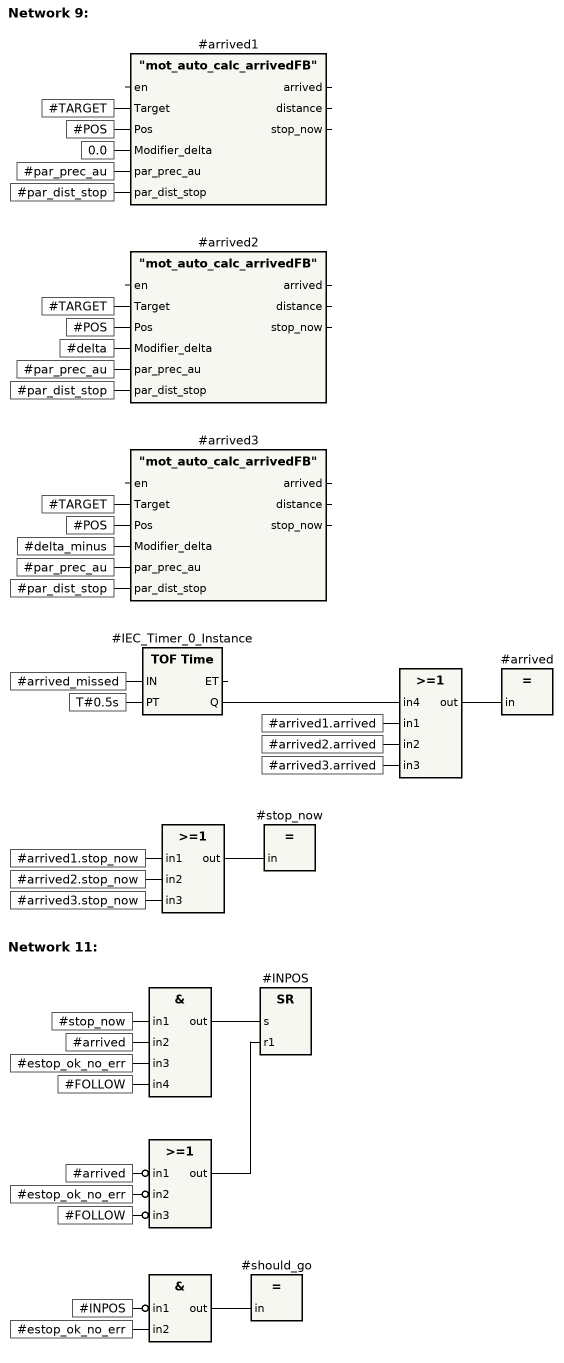
   #arrived1(Target := #TARGET,   // "mot_auto_calc_arrivedFB"
             Pos := #POS,
             Modifier_delta := 0.0,
             par_prec_au := #par_prec_au,
             par_dist_stop := #par_dist_stop);
   #arrived2(Target := #TARGET,   // "mot_auto_calc_arrivedFB"
             Pos := #POS,
             Modifier_delta := #delta,
             par_prec_au := #par_prec_au,
             par_dist_stop := #par_dist_stop);
   #arrived3(Target := #TARGET,   // "mot_auto_calc_arrivedFB"
             Pos := #POS,
             Modifier_delta := #delta_minus,
             par_prec_au := #par_prec_au,
             par_dist_stop := #par_dist_stop);
   #IEC_Timer_0_Instance(IN := #arrived_missed, PT := T#0.5s);   // TOF
   #arrived := #IEC_Timer_0_Instance.Q OR #arrived1.arrived OR #arrived2.arrived OR #arrived3.arrived;
   #stop_now := #arrived1.stop_now OR #arrived2.stop_now OR #arrived3.stop_now;
END_REGION

REGION Network 11
   IF #stop_now AND #arrived AND #estop_ok_no_err AND #FOLLOW THEN
       #INPOS := TRUE;   // SR flip-flop
   END_IF;
   IF NOT #arrived OR NOT #estop_ok_no_err OR NOT #FOLLOW THEN #INPOS := FALSE; END_IF;
   #should_go := NOT #INPOS AND #estop_ok_no_err;
END_REGION

REGION Network 12
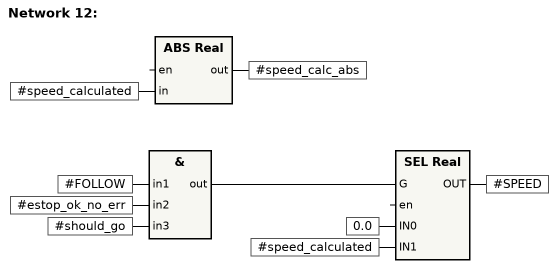
   #speed_calc_abs := ABS(#speed_calculated);
   #SPEED := SEL(G := #FOLLOW AND #estop_ok_no_err AND #should_go, IN0 := 0.0, IN1 := #speed_calculated);
END_REGION
END_FUNCTION_BLOCK

FUNCTION_BLOCK "mot_auto_calc_arrivedFB"   // FB57, FBD
{ S7_Optimized_Access := 'TRUE' }
VERSION : 0.1
// stored: AutoNumber true, IsIECCheckEnabled false, IsRetainMemResEnabled false, MemoryReserve 100, SetENOAutomatically false, UDAEnableTagReadback false
   VAR_INPUT
      Target { ExternalAccessible := 'False'; ExternalVisible := 'False'; ExternalWritable := 'False'} : Real;
      Pos { ExternalAccessible := 'False'; ExternalVisible := 'False'; ExternalWritable := 'False'} : Real;
      Modifier_delta { ExternalAccessible := 'False'; ExternalVisible := 'False'; ExternalWritable := 'False'} : Real;
      par_prec_au { ExternalAccessible := 'False'; ExternalVisible := 'False'; ExternalWritable := 'False'} : Real;
      par_dist_stop { ExternalAccessible := 'False'; ExternalVisible := 'False'; ExternalWritable := 'False'} : Real;
   END_VAR
   VAR_OUTPUT
      arrived { ExternalAccessible := 'False'; ExternalVisible := 'False'; ExternalWritable := 'False'} : Bool;
      distance { ExternalAccessible := 'False'; ExternalVisible := 'False'; ExternalWritable := 'False'} : Real;
      stop_now { ExternalAccessible := 'False'; ExternalVisible := 'False'; ExternalWritable := 'False'} : Bool;
   END_VAR
BEGIN

REGION Network 2 (SCL)
   #distance := #Target - (#Pos + #Modifier_delta);

   #arrived := ABS(#distance) <= #par_prec_au;

   #stop_now := ABS(#distance) <= #par_dist_stop;
END_REGION
END_FUNCTION_BLOCK

FUNCTION_BLOCK "mot_speed_abs_slowly_accelerated"   // FB67, FBD
{ S7_Optimized_Access := 'TRUE' }
VERSION : 0.1
// stored: AutoNumber true, IsIECCheckEnabled false, IsRetainMemResEnabled false, MemoryReserve 100, SetENOAutomatically false, UDAEnableTagReadback false
   VAR_INPUT
      ALLOWED : Bool;
      set_speed_abs : Real;
      v_absMax : Real;
      t_acc : Real;
   END_VAR
   VAR_OUTPUT
      speed_accelerated_slowly_abs : Real;
   END_VAR
   VAR_TEMP
      cycle_time_s : Real;
      acceleration : Real;
      accleration_per_cycle : Real;
   END_VAR
BEGIN

REGION Network 2 (SCL)
   #cycle_time_s := "_MAIN_DB".CLOCK_S_P_SCAN;
   IF #t_acc > 0 THEN
       #acceleration := #v_absMax / #t_acc;
       #accleration_per_cycle := #acceleration * #cycle_time_s;
       IF NOT #ALLOWED OR #set_speed_abs = 0 THEN
           #speed_accelerated_slowly_abs := #set_speed_abs;
       ELSE
           #speed_accelerated_slowly_abs := LIMIT(MN := 0, IN := #speed_accelerated_slowly_abs + #accleration_per_cycle, MX := #set_speed_abs);
       END_IF;
   ELSE
       #speed_accelerated_slowly_abs := #set_speed_abs;
   END_IF;
END_REGION
END_FUNCTION_BLOCK

FUNCTION_BLOCK "mot_speed_wdir_slowly_accelerated"   // FB68, FBD
{ S7_Optimized_Access := 'TRUE' }
VERSION : 0.1
// stored: AutoNumber true, IsIECCheckEnabled false, IsRetainMemResEnabled false, MemoryReserve 100, SetENOAutomatically false, UDAEnableTagReadback false
   VAR_INPUT
      ALLOWED : Bool;
      set_speed__wdir : Real;
      v_absMax : Real;
      t_acc : Real;
      STOP_NOW : Bool;
   END_VAR
   VAR_OUTPUT
      speed_accelerated_slowly_wdir : Real;
   END_VAR
   VAR
      speed_is_zero : Bool;
      speed_is_zero_was : Bool;
      speed_is_zero_CLK : Bool;
   END_VAR
   VAR_TEMP
      cycle_time_s : Real;
      acceleration : Real;
      accleration_per_cycle : Real;
   END_VAR
BEGIN

REGION Network 2 (SCL)
   #speed_is_zero := #set_speed__wdir = 0;
   #speed_is_zero_CLK := false;//AND #speed_is_zero AND NOT #speed_is_zero_was; 
   #speed_is_zero_was := #speed_is_zero ;
END_REGION

REGION Network 3 (SCL)
   #cycle_time_s := "_MAIN_DB".CLOCK_S_P_SCAN;
   IF #t_acc > 0 AND NOT #STOP_NOW THEN
       #acceleration := #v_absMax / #t_acc;
       #accleration_per_cycle := #acceleration * #cycle_time_s;
       IF NOT #ALLOWED OR #speed_is_zero_CLK  THEN
           #speed_accelerated_slowly_wdir := #set_speed__wdir;
       ELSE
           IF #speed_accelerated_slowly_wdir < #set_speed__wdir THEN
               #speed_accelerated_slowly_wdir := MIN(IN1 := #speed_accelerated_slowly_wdir + #accleration_per_cycle, IN2 := #set_speed__wdir);
           ELSE 
               #speed_accelerated_slowly_wdir := MAX(IN1 := #speed_accelerated_slowly_wdir - #accleration_per_cycle,IN2 := #set_speed__wdir);
           END_IF;
       END_IF;
   ELSE
       #speed_accelerated_slowly_wdir := #set_speed__wdir;
   END_IF;
END_REGION
END_FUNCTION_BLOCK

FUNCTION_BLOCK "manual_analog"   // FB7, FBD
{ S7_Optimized_Access := 'TRUE' }
VERSION : 0.1
// stored: AutoNumber true, IsIECCheckEnabled false, IsRetainMemResEnabled false, MemoryReserve 100, SetENOAutomatically false, UDAEnableTagReadback false
   VAR_INPUT
      ALLOWED : Bool;
      ALLOWED_ONLY_IN_OVERRIDE : Bool;
      OVERRIDE_NOW : Bool;
      isMultiturn : Bool;
      POS : Real;
      SET_SPEED : Real;
      xFwdOk : Bool;
      xRevOk : Bool;
      clibrated : Bool;
      par_spd_absmax : Real := 1000.0;
      par_dist_absmax : Real := 100.0;
      par_speed_crawl : Real;
      par_dist_crawl : Real;
      par_dist_stop : Real := 10.0;
      par_spd_blind : Real := 500.0;
      par_fwd_limit : Real := 10000.0;
      par_rev_limit : Real := 0.0;
      par_t_acc : Real;
   END_VAR
   VAR_OUTPUT
      SPEED : Real;
      ER_settings : Bool;
      er_ws : WString;
   END_VAR
   VAR
      speed_slowly_accelerated : Real;
      mot_speed_wdir_slowly_accelerated_Instance { S7_SetPoint := 'True'} : "mot_speed_wdir_slowly_accelerated";
   END_VAR
   VAR_TEMP
      speed_calculated : Real;
      speed_calc_abs : Real;
      estop_ok_no_err : Bool;
      blind : Bool;
      set_spd_loc : Real;
   END_VAR
   VAR CONSTANT
      erwsnoer : WString := WSTRING#'no er';
      erws1 : WString := WSTRING#'lim fwd = rev';
      erws2 : WString := WSTRING#'#par_dist_fast 0';
      erws3 : WString := WSTRING#'#par_spd_absmax';
   END_VAR
   VAR_TEMP   // added for the SCL form of the ladder/FBD networks
      _w1 : Bool;
      _w2 : Bool;
   END_VAR
BEGIN

REGION Network 1
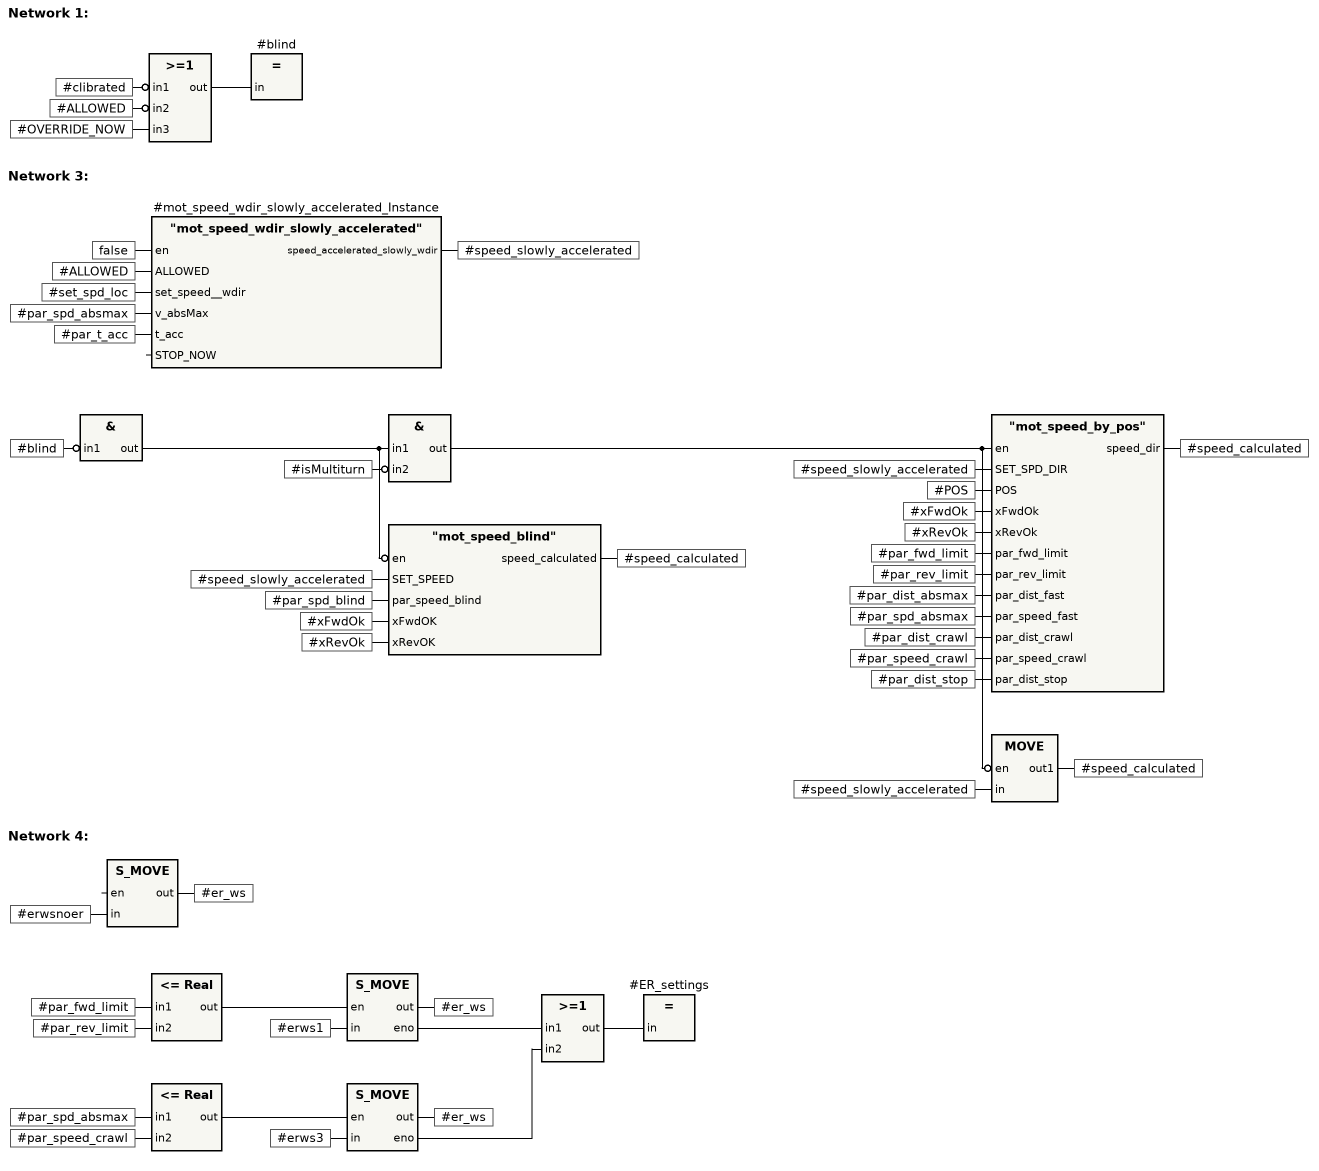
   #blind := NOT #clibrated OR NOT #ALLOWED OR #OVERRIDE_NOW;
END_REGION

REGION Network 2 (SCL)
   #speed_slowly_accelerated := #set_spd_loc := LIMIT(IN:=#SET_SPEED,MN:=-#par_spd_absmax,MX:=#par_spd_absmax);
   //#SET_SPEED*#par_spd_fast
END_REGION

REGION Network 3
   IF false THEN
       #mot_speed_wdir_slowly_accelerated_Instance(ALLOWED := #ALLOWED,   // "mot_speed_wdir_slowly_accelerated"
                               set_speed__wdir := #set_spd_loc,
                               v_absMax := #par_spd_absmax,
                               t_acc := #par_t_acc,
                               speed_accelerated_slowly_wdir => #speed_slowly_accelerated);
   END_IF;
   #_w1 := NOT #blind AND NOT #isMultiturn;
   IF #_w1 THEN
       "mot_speed_by_pos"(SET_SPD_DIR := #speed_slowly_accelerated,
                          POS := #POS,
                          xFwdOk := #xFwdOk,
                          xRevOk := #xRevOk,
                          par_fwd_limit := #par_fwd_limit,
                          par_rev_limit := #par_rev_limit,
                          par_dist_fast := #par_dist_absmax,
                          par_speed_fast := #par_spd_absmax,
                          par_dist_crawl := #par_dist_crawl,
                          par_speed_crawl := #par_speed_crawl,
                          par_dist_stop := #par_dist_stop,
                          speed_dir => #speed_calculated);
   END_IF;
   IF NOT #_w1 THEN #speed_calculated := #speed_slowly_accelerated; END_IF;
   IF NOT (NOT #blind) THEN
       "mot_speed_blind"(SET_SPEED := #speed_slowly_accelerated,
                         par_speed_blind := #par_spd_blind,
                         xFwdOK := #xFwdOk,
                         xRevOK := #xRevOk,
                         speed_calculated => #speed_calculated);
   END_IF;
END_REGION

REGION Network 4
   #er_ws := #erwsnoer;
   #_w1 := #par_fwd_limit <= #par_rev_limit;
   IF #_w1 THEN #er_ws := #erws1; END_IF;
   #_w2 := #par_spd_absmax <= #par_speed_crawl;
   IF #_w2 THEN #er_ws := #erws3; END_IF;
   #ER_settings := #_w1 OR #_w2;
END_REGION

REGION Network 5
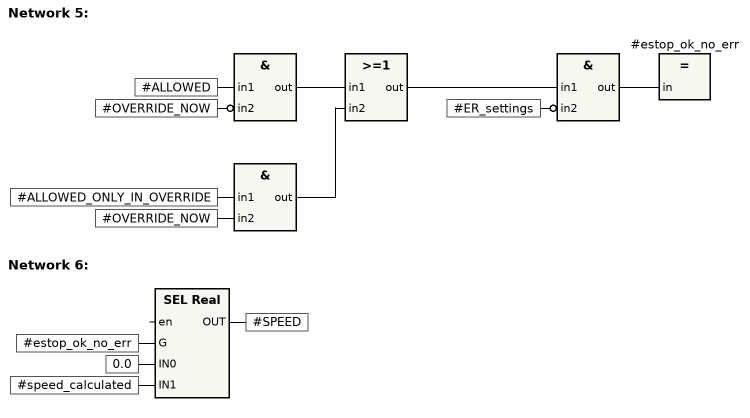
   #estop_ok_no_err := ((#ALLOWED AND NOT #OVERRIDE_NOW) OR (#ALLOWED_ONLY_IN_OVERRIDE AND #OVERRIDE_NOW)) AND NOT #ER_settings;
END_REGION

REGION Network 6
   #SPEED := SEL(G := #estop_ok_no_err, IN0 := 0.0, IN1 := #speed_calculated);
END_REGION
END_FUNCTION_BLOCK

FUNCTION "mot_speed_blind" : Void   // FC11, FBD
{ S7_Optimized_Access := 'TRUE' }
VERSION : 0.1
// stored: AutoNumber true, IsIECCheckEnabled false, SetENOAutomatically false, UDAEnableTagReadback false
   VAR_INPUT
      SET_SPEED : Real;
      par_speed_blind : Real;
      xFwdOK : Bool;
      xRevOK : Bool;
   END_VAR
   VAR_OUTPUT
      speed_calculated : Real;
   END_VAR
   VAR_TEMP
      go_fwd : Bool;
      go_rev : Bool;
   END_VAR
BEGIN

REGION Network 1
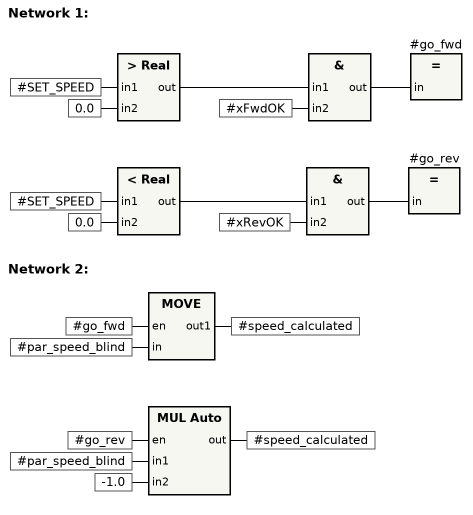
   #go_fwd := (#SET_SPEED > 0.0) AND #xFwdOK;
   #go_rev := (#SET_SPEED < 0.0) AND #xRevOK;
END_REGION

REGION Network 2
   IF #go_fwd THEN #speed_calculated := #par_speed_blind; END_IF;
   IF #go_rev THEN #speed_calculated := #par_speed_blind * (-1.0); END_IF;
END_REGION
END_FUNCTION

FUNCTION_BLOCK "enc_no_change_in_time"   // FB6, FBD
{ S7_Optimized_Access := 'TRUE' }
VERSION : 0.1
// stored: AutoNumber true, IsIECCheckEnabled false, IsRetainMemResEnabled false, MemoryReserve 100, SetENOAutomatically false, UDAEnableTagReadback false
   VAR_INPUT
      pt : Time := T#1s;
      FWD : Bool;
      REV : Bool;
      POS : Real;
   END_VAR
   VAR_OUTPUT
      ER_FWD : Bool;
      ER_REV : Bool;
   END_VAR
   VAR
      going_fwd { ExternalAccessible := 'False'; ExternalVisible := 'False'; ExternalWritable := 'False'} : Bool;
      going_rev { ExternalAccessible := 'False'; ExternalVisible := 'False'; ExternalWritable := 'False'} : Bool;
      going_not { ExternalAccessible := 'False'; ExternalVisible := 'False'; ExternalWritable := 'False'} : Bool;
      mem : Real;
      t_fwd { S7_SetPoint := 'True'} : TON_TIME;
      t_rev { S7_SetPoint := 'True'} : TON_TIME;
   END_VAR
BEGIN

REGION Network 1
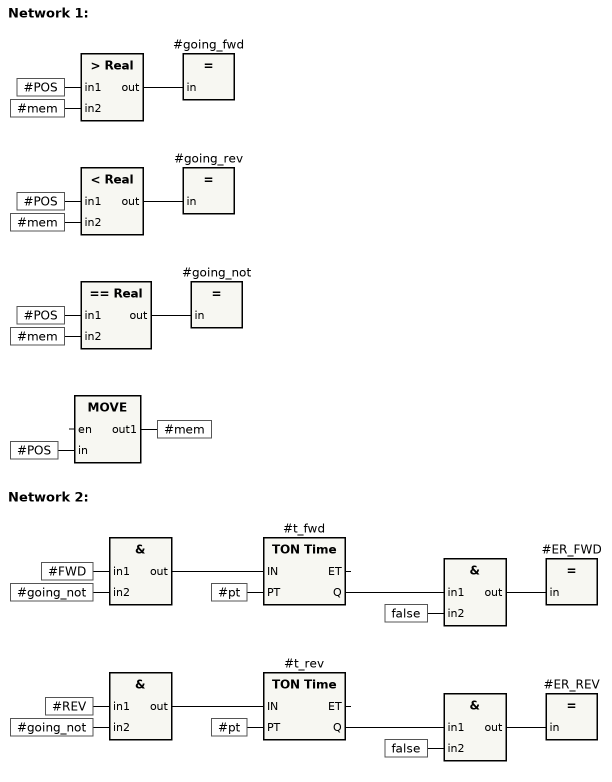
   #going_fwd := #POS > #mem;
   #going_rev := #POS < #mem;
   #going_not := #POS = #mem;
   #mem := #POS;
END_REGION

REGION Network 2
   #t_fwd(IN := #FWD AND #going_not, PT := #pt);   // TON
   #ER_FWD := #t_fwd.Q AND false;
   #t_rev(IN := #REV AND #going_not, PT := #pt);   // TON
   #ER_REV := #t_rev.Q AND false;
END_REGION
END_FUNCTION_BLOCK

FUNCTION_BLOCK "BRK_FB"   // FB21, FBD
{ S7_Optimized_Access := 'TRUE' }
VERSION : 0.1
// stored: AutoNumber true, IsIECCheckEnabled false, IsRetainMemResEnabled false, MemoryReserve 100, SetENOAutomatically false, UDAEnableTagReadback false
   VAR_INPUT
      SpeedZero : Bool;
      fwd : Bool;
      rev : Bool;
      pt : Time := T#100ms;
      error : Bool;
   END_VAR
   VAR_OUTPUT
      BRK_REL { ExternalAccessible := 'False'; ExternalVisible := 'False'; ExternalWritable := 'False'} : Bool;
   END_VAR
   VAR
      IEC_Timer_0_Instance { S7_SetPoint := 'True'} : TOF_TIME;
   END_VAR
BEGIN

REGION Network 2
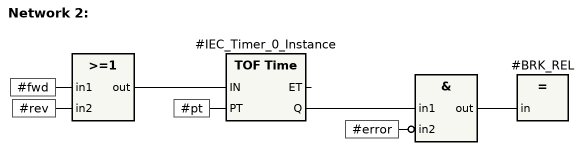
   #IEC_Timer_0_Instance(IN := #fwd OR #rev, PT := #pt);   // TOF
   #BRK_REL := #IEC_Timer_0_Instance.Q AND NOT #error;
END_REGION
END_FUNCTION_BLOCK

FUNCTION "f_ao_10V" : Int
{ S7_Optimized_Access := 'TRUE' }
VERSION : 0.1
   VAR_INPUT 
      "in 0.0-10.0" : Real;
   END_VAR

   VAR_TEMP 
      value_for_10V : Real;
      "r10.0" : Real;
   END_VAR


BEGIN
	#value_for_10V := 27648.0;(* tested FPY value 27175.0 *)
	#"r10.0" := 10.0;
	#f_ao_10V := DINT_TO_INT(
	                                 REAL_TO_DINT(
	                                              LIMIT(IN := #"in 0.0-10.0", MN := 0, MX := #"r10.0")
	                                              / #"r10.0" * #value_for_10V)
	);
END_FUNCTION

ORGANIZATION_BLOCK "Cyclic interrupt_axis_30ms"   // OB31, LAD, CyclicInterrupt
{ S7_Optimized_Access := 'TRUE' }
VERSION : 0.1
// stored: AutoNumber true, IsIECCheckEnabled false, SetENOAutomatically false
   VAR_INPUT
      Initial_Call : Bool;
      Event_Count : Int;
   END_VAR
BEGIN

REGION Network 1
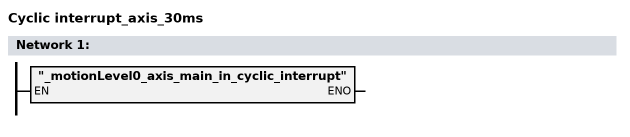
   RUNG wire#powerrail
      "_motionLevel0_axis_main_in_cyclic_interrupt"()
   END_RUNG
   // the same network as SCL:
   "_motionLevel0_axis_main_in_cyclic_interrupt"();
END_REGION
END_ORGANIZATION_BLOCK

FUNCTION "_motionLevel0_axis_main_in_cyclic_interrupt" : Void   // FC13, FBD
{ S7_Optimized_Access := 'TRUE' }
VERSION : 0.1
// stored: AutoNumber true, IsIECCheckEnabled false, SetENOAutomatically false, UDAEnableTagReadback false
   VAR_TEMP
      doors : Bool;
      "xray uses doors fwd closed mech" : Bool;
      "добавить блокировку вперед по световой завесе" : Bool;
      loc_dor_c_opn : Bool;
      loc_dor_c_cls : Bool;
      doorsWnOpnNAld : Bool;
      doorsWnClsNAld : Bool;
      ошибка_задания_искуственных_границ : Bool;
      динамическая_граница_y_rev : Real;
      динамическая_граница_y_fwd : Real;
      динамическая_граница_x_rev : Real;
      динамическая_граница_x_fwd : Real;
      манипулятор_не_мешает_дверям : Bool;
      doors_wnmanipulator : Bool;
   END_VAR
BEGIN

REGION Network 2
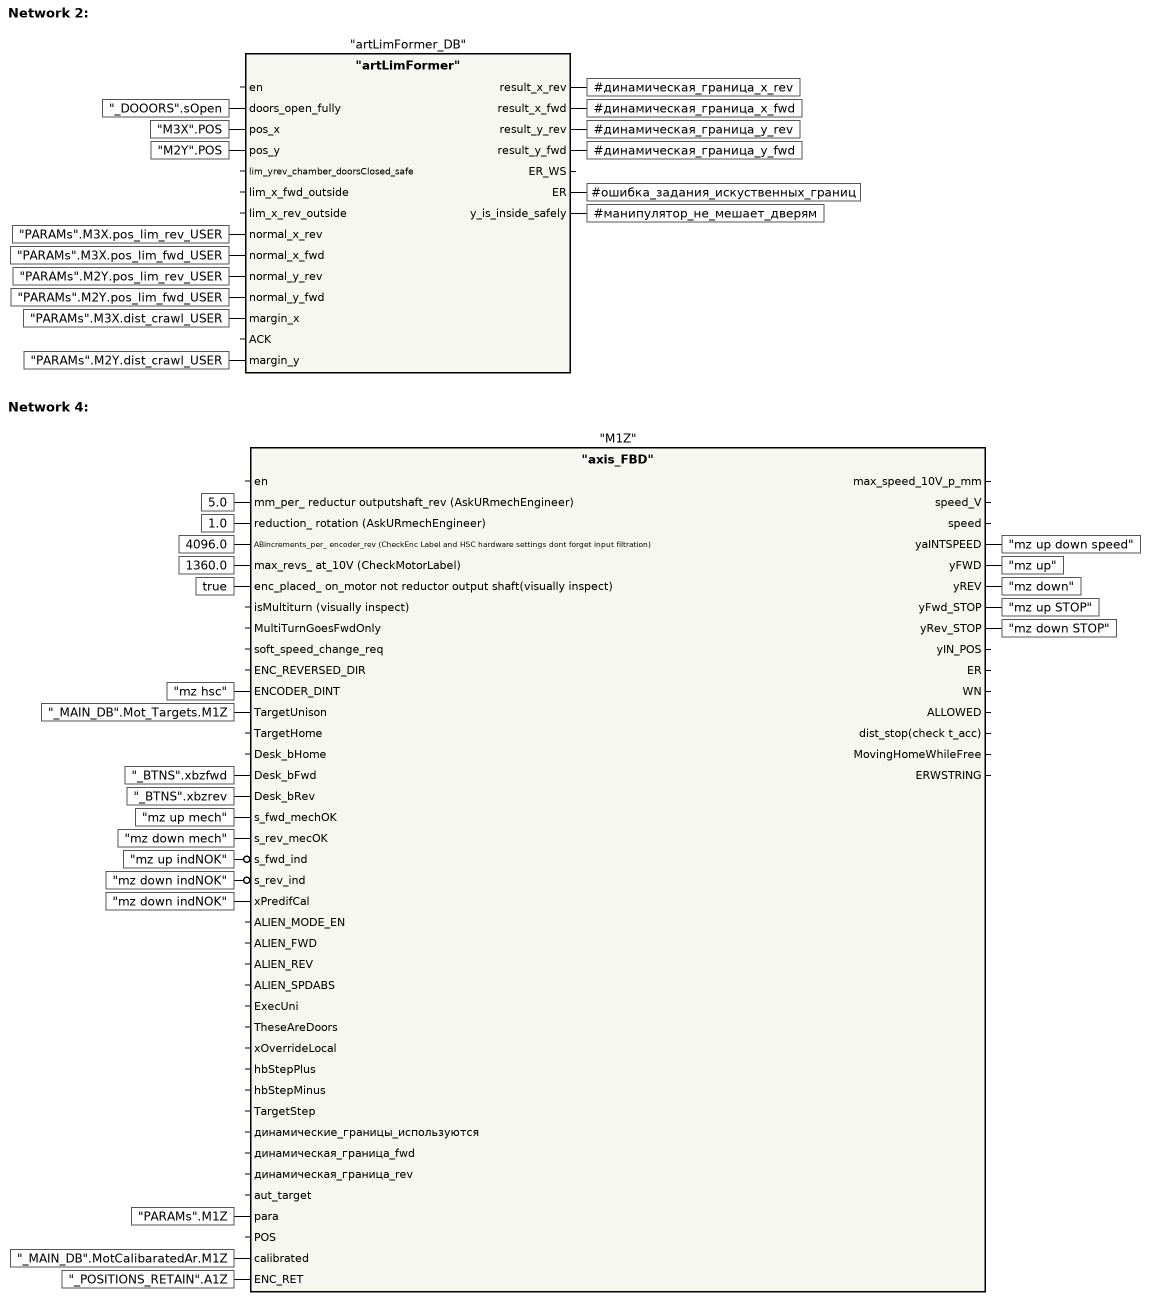
   "artLimFormer_DB"(doors_open_fully := "_DOOORS".sOpen,   // "artLimFormer"
                     pos_x := "M3X".POS,
                     pos_y := "M2Y".POS,
                     normal_x_rev := "PARAMs".M3X.pos_lim_rev_USER,
                     normal_x_fwd := "PARAMs".M3X.pos_lim_fwd_USER,
                     normal_y_rev := "PARAMs".M2Y.pos_lim_rev_USER,
                     normal_y_fwd := "PARAMs".M2Y.pos_lim_fwd_USER,
                     margin_x := "PARAMs".M3X.dist_crawl_USER,
                     margin_y := "PARAMs".M2Y.dist_crawl_USER,
                     result_x_rev => #динамическая_граница_x_rev,
                     result_x_fwd => #динамическая_граница_x_fwd,
                     result_y_rev => #динамическая_граница_y_rev,
                     result_y_fwd => #динамическая_граница_y_fwd,
                     ER => #ошибка_задания_искуственных_границ,
                     y_is_inside_safely => #манипулятор_не_мешает_дверям);
END_REGION

REGION Network 4
   "M1Z"("mm_per_ reductur outputshaft_rev (AskURmechEngineer)" := 5.0,   // "axis_FBD"
         "reduction_ rotation (AskURmechEngineer)" := 1.0,
         "ABincrements_per_ encoder_rev (CheckEnc Label and HSC hardware settings dont forget input filtration)" := 4096.0,
         "max_revs_ at_10V (CheckMotorLabel)" := 1360.0,
         "enc_placed_ on_motor not reductor output shaft(visually inspect)" := true,
         ENCODER_DINT := "mz hsc",
         TargetUnison := "_MAIN_DB".Mot_Targets.M1Z,
         Desk_bFwd := "_BTNS".xbzfwd,
         Desk_bRev := "_BTNS".xbzrev,
         s_fwd_mechOK := "mz up mech",
         s_rev_mecOK := "mz down mech",
         s_fwd_ind := NOT "mz up indNOK",
         s_rev_ind := NOT "mz down indNOK",
         xPredifCal := "mz down indNOK",
         para := "PARAMs".M1Z,
         calibrated := "_MAIN_DB".MotCalibaratedAr.M1Z,
         ENC_RET := "_POSITIONS_RETAIN".A1Z,
         yaINTSPEED => "mz up down speed",
         yFWD => "mz up",
         yREV => "mz down",
         yFwd_STOP => "mz up STOP",
         yRev_STOP => "mz down STOP");
END_REGION

REGION Network 5
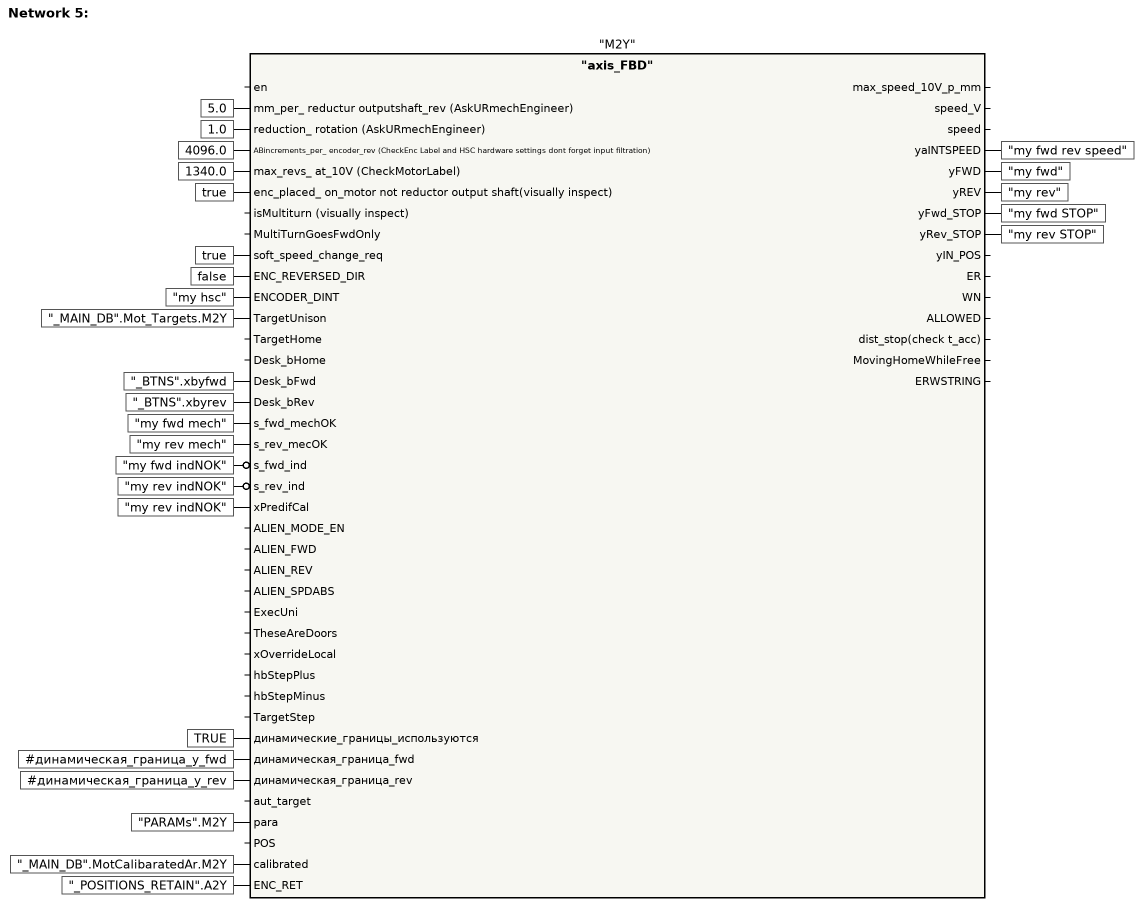
   "M2Y"("mm_per_ reductur outputshaft_rev (AskURmechEngineer)" := 5.0,   // "axis_FBD"
         "reduction_ rotation (AskURmechEngineer)" := 1.0,
         "ABincrements_per_ encoder_rev (CheckEnc Label and HSC hardware settings dont forget input filtration)" := 4096.0,
         "max_revs_ at_10V (CheckMotorLabel)" := 1340.0,
         "enc_placed_ on_motor not reductor output shaft(visually inspect)" := true,
         soft_speed_change_req := true,
         ENC_REVERSED_DIR := false,
         ENCODER_DINT := "my hsc",
         TargetUnison := "_MAIN_DB".Mot_Targets.M2Y,
         Desk_bFwd := "_BTNS".xbyfwd,
         Desk_bRev := "_BTNS".xbyrev,
         s_fwd_mechOK := "my fwd mech",
         s_rev_mecOK := "my rev mech",
         s_fwd_ind := NOT "my fwd indNOK",
         s_rev_ind := NOT "my rev indNOK",
         xPredifCal := "my rev indNOK",
         динамические_границы_используются := TRUE,
         динамическая_граница_fwd := #динамическая_граница_y_fwd,
         динамическая_граница_rev := #динамическая_граница_y_rev,
         para := "PARAMs".M2Y,
         calibrated := "_MAIN_DB".MotCalibaratedAr.M2Y,
         ENC_RET := "_POSITIONS_RETAIN".A2Y,
         yaINTSPEED => "my fwd rev speed",
         yFWD => "my fwd",
         yREV => "my rev",
         yFwd_STOP => "my fwd STOP",
         yRev_STOP => "my rev STOP");
END_REGION

REGION Network 6
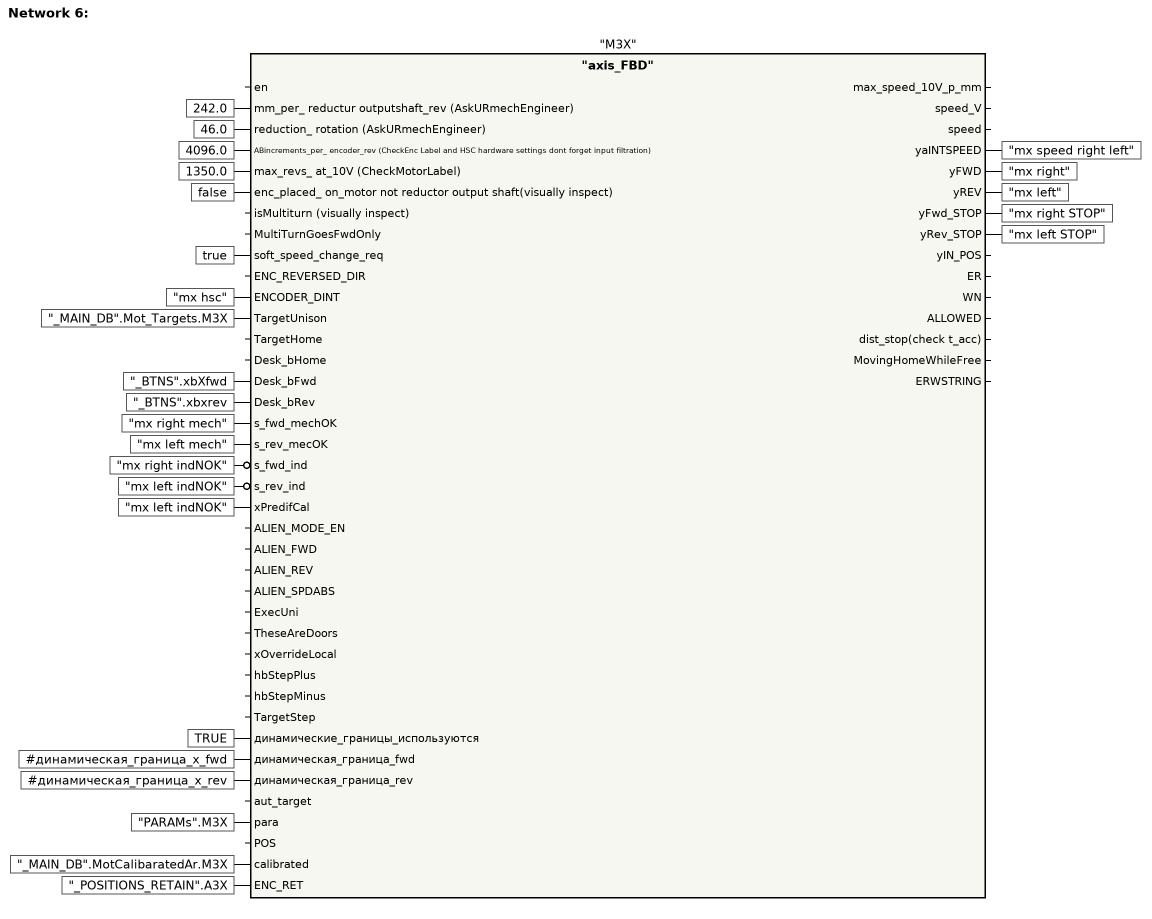
   "M3X"("mm_per_ reductur outputshaft_rev (AskURmechEngineer)" := 242.0,   // "axis_FBD"
         "reduction_ rotation (AskURmechEngineer)" := 46.0,
         "ABincrements_per_ encoder_rev (CheckEnc Label and HSC hardware settings dont forget input filtration)" := 4096.0,
         "max_revs_ at_10V (CheckMotorLabel)" := 1350.0,
         "enc_placed_ on_motor not reductor output shaft(visually inspect)" := false,
         soft_speed_change_req := true,
         ENCODER_DINT := "mx hsc",
         TargetUnison := "_MAIN_DB".Mot_Targets.M3X,
         Desk_bFwd := "_BTNS".xbXfwd,
         Desk_bRev := "_BTNS".xbxrev,
         s_fwd_mechOK := "mx right mech",
         s_rev_mecOK := "mx left mech",
         s_fwd_ind := NOT "mx right indNOK",
         s_rev_ind := NOT "mx left indNOK",
         xPredifCal := "mx left indNOK",
         динамические_границы_используются := TRUE,
         динамическая_граница_fwd := #динамическая_граница_x_fwd,
         динамическая_граница_rev := #динамическая_граница_x_rev,
         para := "PARAMs".M3X,
         calibrated := "_MAIN_DB".MotCalibaratedAr.M3X,
         ENC_RET := "_POSITIONS_RETAIN".A3X,
         yaINTSPEED => "mx speed right left",
         yFWD => "mx right",
         yREV => "mx left",
         yFwd_STOP => "mx right STOP",
         yRev_STOP => "mx left STOP");
END_REGION

REGION Network 7
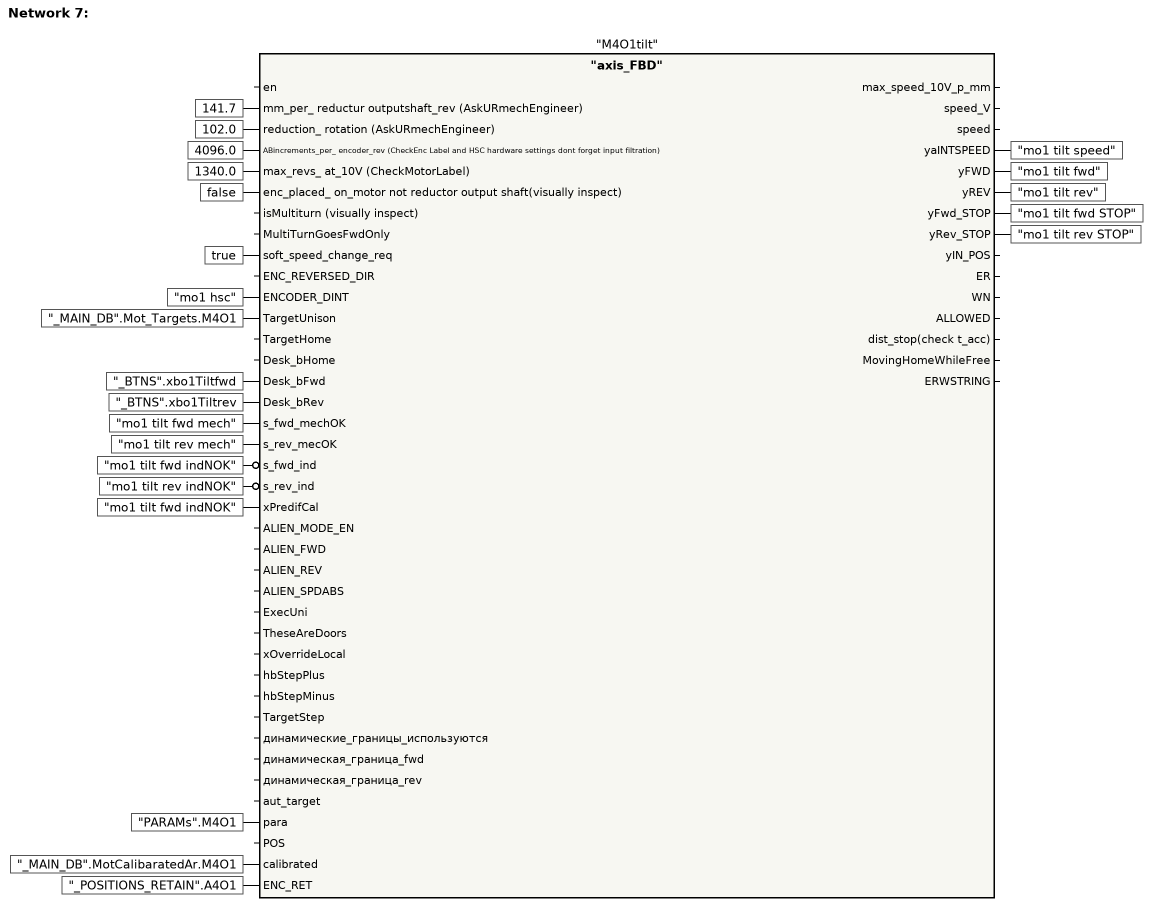
   "M4O1tilt"("mm_per_ reductur outputshaft_rev (AskURmechEngineer)" := 141.7,   // "axis_FBD"
              "reduction_ rotation (AskURmechEngineer)" := 102.0,
              "ABincrements_per_ encoder_rev (CheckEnc Label and HSC hardware settings dont forget input filtration)" := 4096.0,
              "max_revs_ at_10V (CheckMotorLabel)" := 1340.0,
              "enc_placed_ on_motor not reductor output shaft(visually inspect)" := false,
              soft_speed_change_req := true,
              ENCODER_DINT := "mo1 hsc",
              TargetUnison := "_MAIN_DB".Mot_Targets.M4O1,
              Desk_bFwd := "_BTNS".xbo1Tiltfwd,
              Desk_bRev := "_BTNS".xbo1Tiltrev,
              s_fwd_mechOK := "mo1 tilt fwd mech",
              s_rev_mecOK := "mo1 tilt rev mech",
              s_fwd_ind := NOT "mo1 tilt fwd indNOK",
              s_rev_ind := NOT "mo1 tilt rev indNOK",
              xPredifCal := "mo1 tilt fwd indNOK",
              para := "PARAMs".M4O1,
              calibrated := "_MAIN_DB".MotCalibaratedAr.M4O1,
              ENC_RET := "_POSITIONS_RETAIN".A4O1,
              yaINTSPEED => "mo1 tilt speed",
              yFWD => "mo1 tilt fwd",
              yREV => "mo1 tilt rev",
              yFwd_STOP => "mo1 tilt fwd STOP",
              yRev_STOP => "mo1 tilt rev STOP");
END_REGION

REGION Network 8
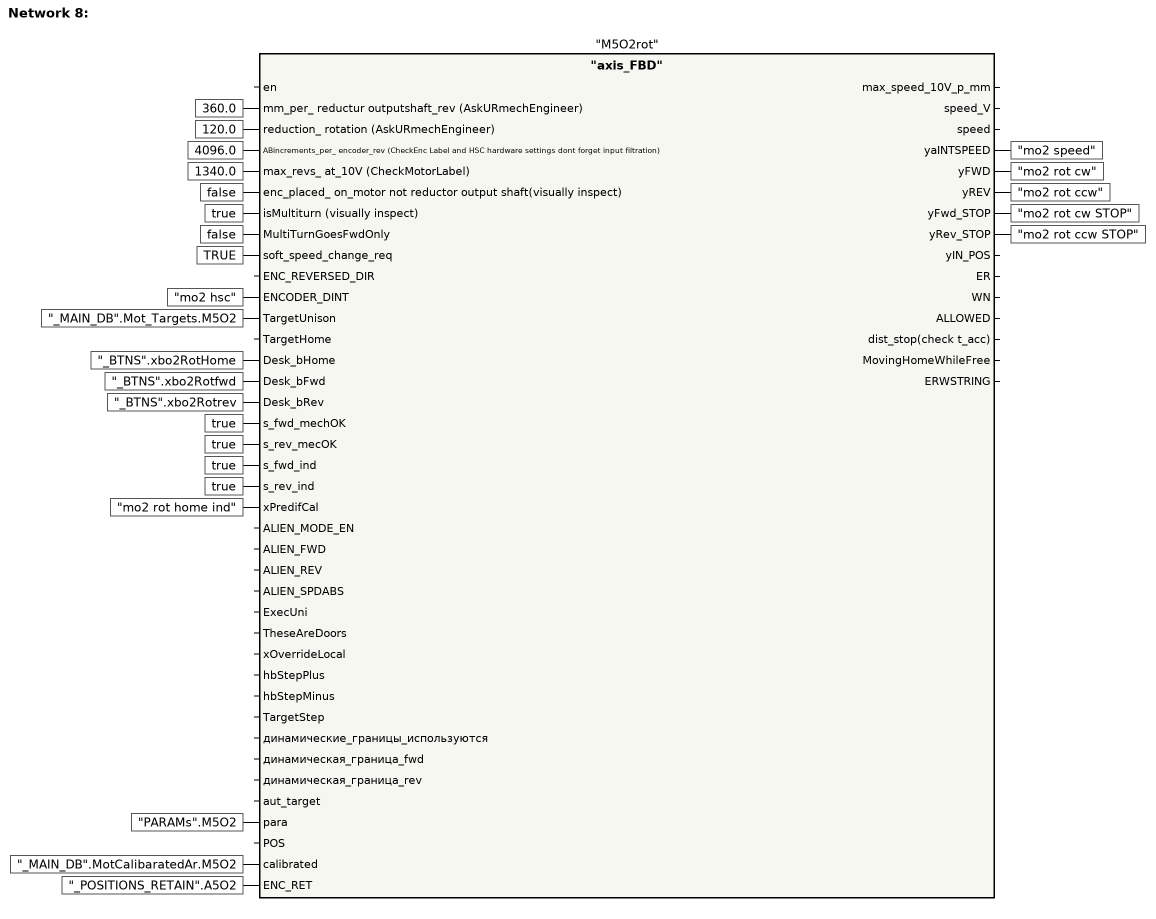
   "M5O2rot"("mm_per_ reductur outputshaft_rev (AskURmechEngineer)" := 360.0,   // "axis_FBD"
             "reduction_ rotation (AskURmechEngineer)" := 120.0,
             "ABincrements_per_ encoder_rev (CheckEnc Label and HSC hardware settings dont forget input filtration)" := 4096.0,
             "max_revs_ at_10V (CheckMotorLabel)" := 1340.0,
             "enc_placed_ on_motor not reductor output shaft(visually inspect)" := false,
             "isMultiturn (visually inspect)" := true,
             MultiTurnGoesFwdOnly := false,
             soft_speed_change_req := TRUE,
             ENCODER_DINT := "mo2 hsc",
             TargetUnison := "_MAIN_DB".Mot_Targets.M5O2,
             Desk_bHome := "_BTNS".xbo2RotHome,
             Desk_bFwd := "_BTNS".xbo2Rotfwd,
             Desk_bRev := "_BTNS".xbo2Rotrev,
             s_fwd_mechOK := true,
             s_rev_mecOK := true,
             s_fwd_ind := true,
             s_rev_ind := true,
             xPredifCal := "mo2 rot home ind",
             para := "PARAMs".M5O2,
             calibrated := "_MAIN_DB".MotCalibaratedAr.M5O2,
             ENC_RET := "_POSITIONS_RETAIN".A5O2,
             yaINTSPEED => "mo2 speed",
             yFWD => "mo2 rot cw",
             yREV => "mo2 rot ccw",
             yFwd_STOP => "mo2 rot cw STOP",
             yRev_STOP => "mo2 rot ccw STOP");
END_REGION

REGION Network 9
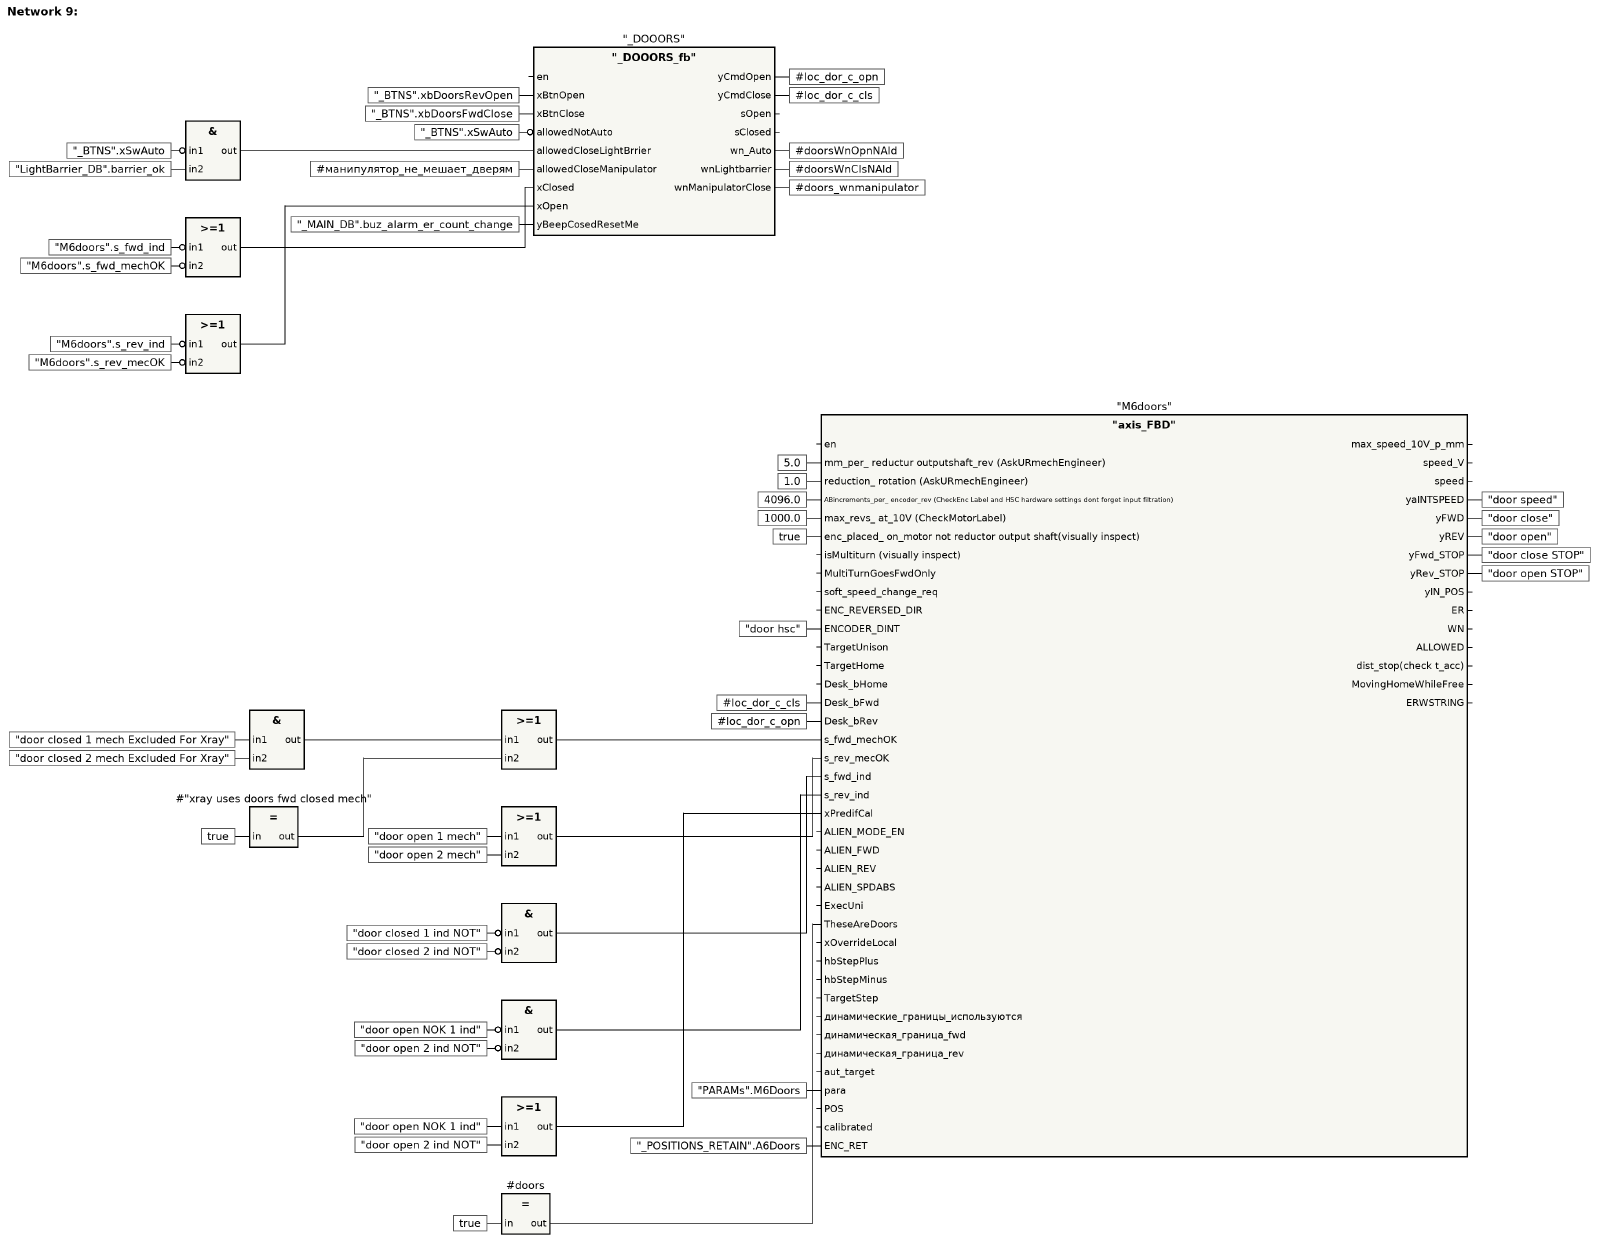
   "_DOOORS"(xBtnOpen := "_BTNS".xbDoorsRevOpen,   // "_DOOORS_fb"
             xBtnClose := "_BTNS".xbDoorsFwdClose,
             allowedNotAuto := NOT "_BTNS".xSwAuto,
             allowedCloseLightBrrier := NOT "_BTNS".xSwAuto AND "LightBarrier_DB".barrier_ok,
             allowedCloseManipulator := #манипулятор_не_мешает_дверям,
             xClosed := NOT "M6doors".s_fwd_ind OR NOT "M6doors".s_fwd_mechOK,
             xOpen := NOT "M6doors".s_rev_ind OR NOT "M6doors".s_rev_mecOK,
             yBeepCosedResetMe := "_MAIN_DB".buz_alarm_er_count_change,
             yCmdOpen => #loc_dor_c_opn,
             yCmdClose => #loc_dor_c_cls,
             wn_Auto => #doorsWnOpnNAld,
             wnLightbarrier => #doorsWnClsNAld,
             wnManipulatorClose => #doors_wnmanipulator);
   #"xray uses doors fwd closed mech" := true;
   #doors := true;
   "M6doors"("mm_per_ reductur outputshaft_rev (AskURmechEngineer)" := 5.0,   // "axis_FBD"
             "reduction_ rotation (AskURmechEngineer)" := 1.0,
             "ABincrements_per_ encoder_rev (CheckEnc Label and HSC hardware settings dont forget input filtration)" := 4096.0,
             "max_revs_ at_10V (CheckMotorLabel)" := 1000.0,
             "enc_placed_ on_motor not reductor output shaft(visually inspect)" := true,
             ENCODER_DINT := "door hsc",
             Desk_bFwd := #loc_dor_c_cls,
             Desk_bRev := #loc_dor_c_opn,
             s_fwd_mechOK := ("door closed 1 mech Excluded For Xray" AND "door closed 2 mech Excluded For Xray") OR true,
             s_rev_mecOK := "door open 1 mech" OR "door open 2 mech",
             s_fwd_ind := NOT "door closed 1 ind NOT" AND NOT "door closed 2 ind NOT",
             s_rev_ind := NOT "door open NOK 1 ind" AND NOT "door open 2 ind NOT",
             xPredifCal := "door open NOK 1 ind" OR "door open 2 ind NOT",
             TheseAreDoors := true,
             para := "PARAMs".M6Doors,
             ENC_RET := "_POSITIONS_RETAIN".A6Doors,
             yaINTSPEED => "door speed",
             yFWD => "door close",
             yREV => "door open",
             yFwd_STOP => "door close STOP",
             yRev_STOP => "door open STOP");
END_REGION

REGION Network 10
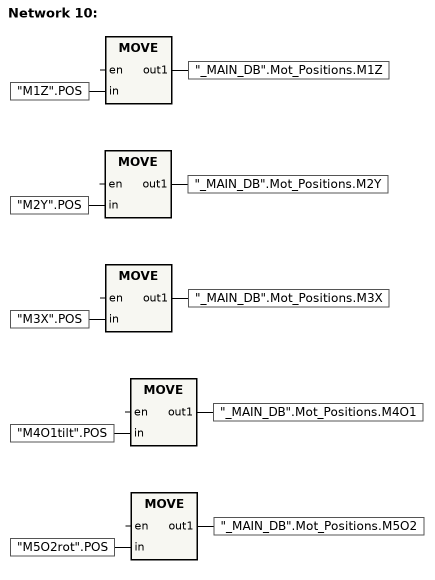
   "_MAIN_DB".Mot_Positions.M1Z := "M1Z".POS;
   "_MAIN_DB".Mot_Positions.M2Y := "M2Y".POS;
   "_MAIN_DB".Mot_Positions.M3X := "M3X".POS;
   "_MAIN_DB".Mot_Positions.M4O1 := "M4O1tilt".POS;
   "_MAIN_DB".Mot_Positions.M5O2 := "M5O2rot".POS;
END_REGION

REGION Network 11
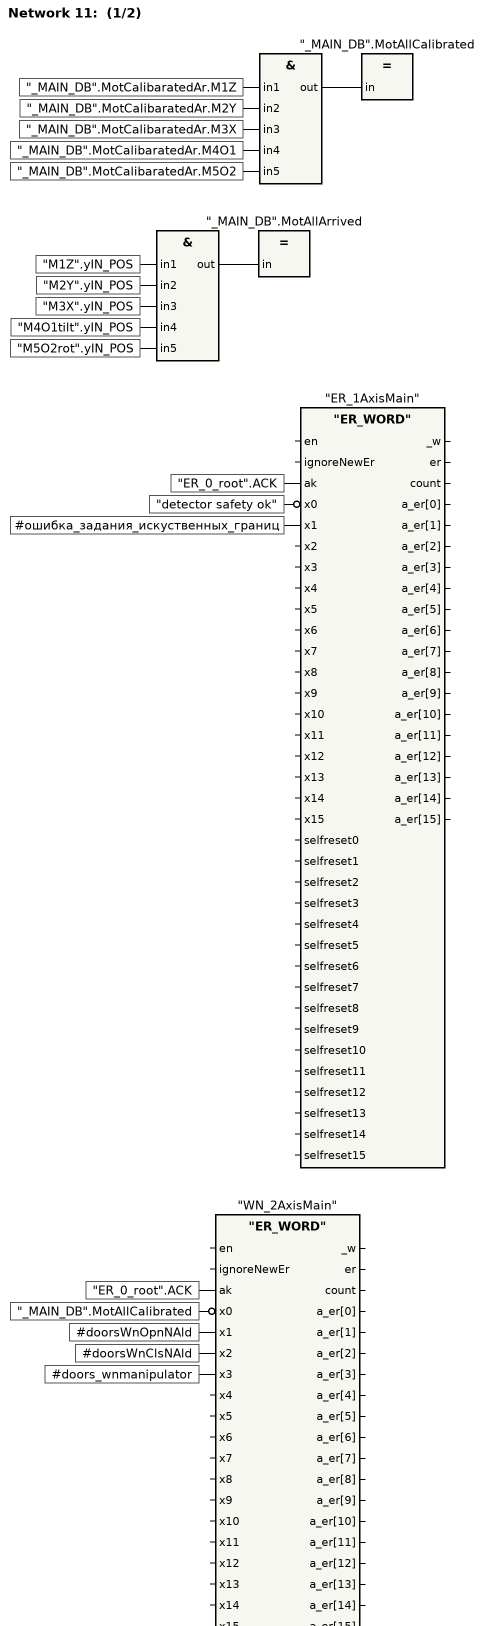
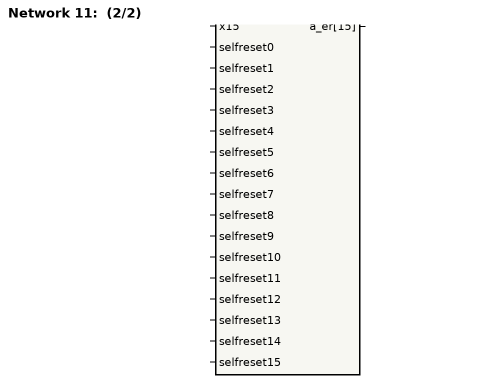
   "_MAIN_DB".MotAllCalibrated := "_MAIN_DB".MotCalibaratedAr.M1Z AND "_MAIN_DB".MotCalibaratedAr.M2Y AND "_MAIN_DB".MotCalibaratedAr.M3X AND "_MAIN_DB".MotCalibaratedAr.M4O1 AND "_MAIN_DB".MotCalibaratedAr.M5O2;
   "_MAIN_DB".MotAllArrived := "M1Z".yIN_POS AND "M2Y".yIN_POS AND "M3X".yIN_POS AND "M4O1tilt".yIN_POS AND "M5O2rot".yIN_POS;
   "ER_1AxisMain"(ak := "ER_0_root".ACK,   // "ER_WORD"
                  x0 := NOT "detector safety ok",
                  x1 := #ошибка_задания_искуственных_границ);
   "WN_2AxisMain"(ak := "ER_0_root".ACK,   // "ER_WORD"
                  x0 := NOT "_MAIN_DB".MotAllCalibrated,
                  x1 := #doorsWnOpnNAld,
                  x2 := #doorsWnClsNAld,
                  x3 := #doors_wnmanipulator);
END_REGION
END_FUNCTION

FUNCTION_BLOCK "artLimFormer"   // FB74, FBD
{ S7_Optimized_Access := 'TRUE' }
VERSION : 0.1
// stored: AutoNumber true, IsIECCheckEnabled false, IsRetainMemResEnabled false, MemoryReserve 100, SetENOAutomatically false, UDAEnableTagReadback false
   VAR_INPUT
      doors_open_fully : Bool;
      pos_x : Real;
      pos_y : Real;
      lim_yrev_chamber_doorsClosed_safe : Real;
      lim_x_fwd_outside : Real;
      lim_x_rev_outside : Real;
      normal_x_rev : Real;
      normal_x_fwd : Real;
      normal_y_rev : Real;
      normal_y_fwd : Real;
      margin_x : Real;
      ACK : Bool;
      margin_y : Real;
   END_VAR
   VAR_OUTPUT
      result_x_rev : Real;
      result_x_fwd : Real;
      result_y_rev : Real;
      result_y_fwd : Real;
      ER_WS : WString;
      ER : Bool;
      y_is_inside_safely : Bool;
   END_VAR
   VAR
      y_can_go_out_rev : Bool;
      x_fits_in_doors : Bool;
      y_is_inside : Bool;
   END_VAR
   VAR_TEMP
      lim_x_fwd_outside_p_margin : Real;
      loc_lim_x_fwd_outside_p_margin : Real;
      loc_lim_x_rev_outside_m_margin : Real;
      loc_lim_yrev_chamber_doorsClosed_safe_m_margin : Real;
   END_VAR
   VAR CONSTANT
      erws1 : WString := WSTRING#'wrong limits';
   END_VAR
BEGIN

REGION Network 1 (SCL)
   #loc_lim_x_fwd_outside_p_margin := #lim_x_fwd_outside + #margin_x;
   #loc_lim_x_rev_outside_m_margin := #lim_x_rev_outside - #margin_x; 

   #loc_lim_yrev_chamber_doorsClosed_safe_m_margin := #lim_yrev_chamber_doorsClosed_safe - #margin_y;
END_REGION

REGION Network 2
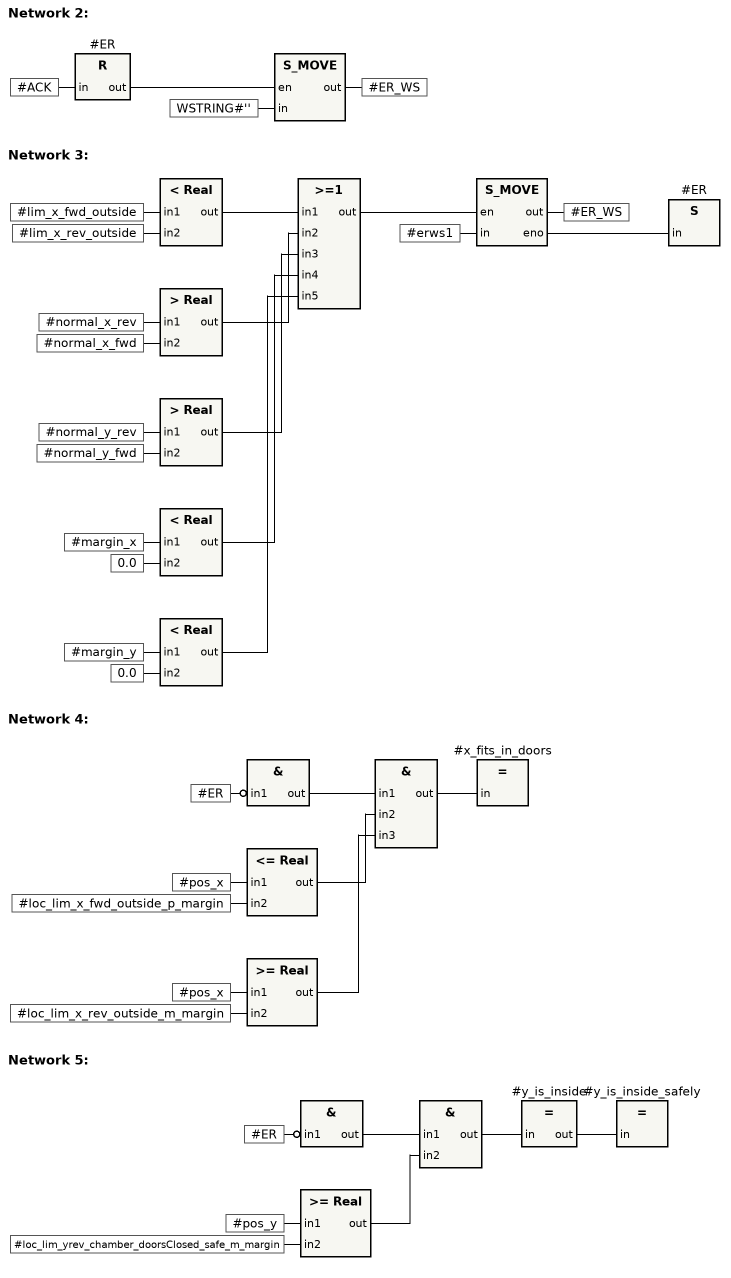
   IF #ACK THEN
       #ER := FALSE;
       #ER_WS := WSTRING#'';
   END_IF;
END_REGION

REGION Network 3
   IF (#lim_x_fwd_outside < #lim_x_rev_outside) OR (#normal_x_rev > #normal_x_fwd) OR (#normal_y_rev > #normal_y_fwd) OR (#margin_x < 0.0) OR (#margin_y < 0.0) THEN
       #ER_WS := #erws1;
       #ER := TRUE;
   END_IF;
END_REGION

REGION Network 4
   #x_fits_in_doors := NOT #ER AND (#pos_x <= #loc_lim_x_fwd_outside_p_margin) AND (#pos_x >= #loc_lim_x_rev_outside_m_margin);
END_REGION

REGION Network 5
   #y_is_inside := NOT #ER AND (#pos_y >= #loc_lim_yrev_chamber_doorsClosed_safe_m_margin);
   #y_is_inside_safely := #y_is_inside;
END_REGION

REGION Network 6
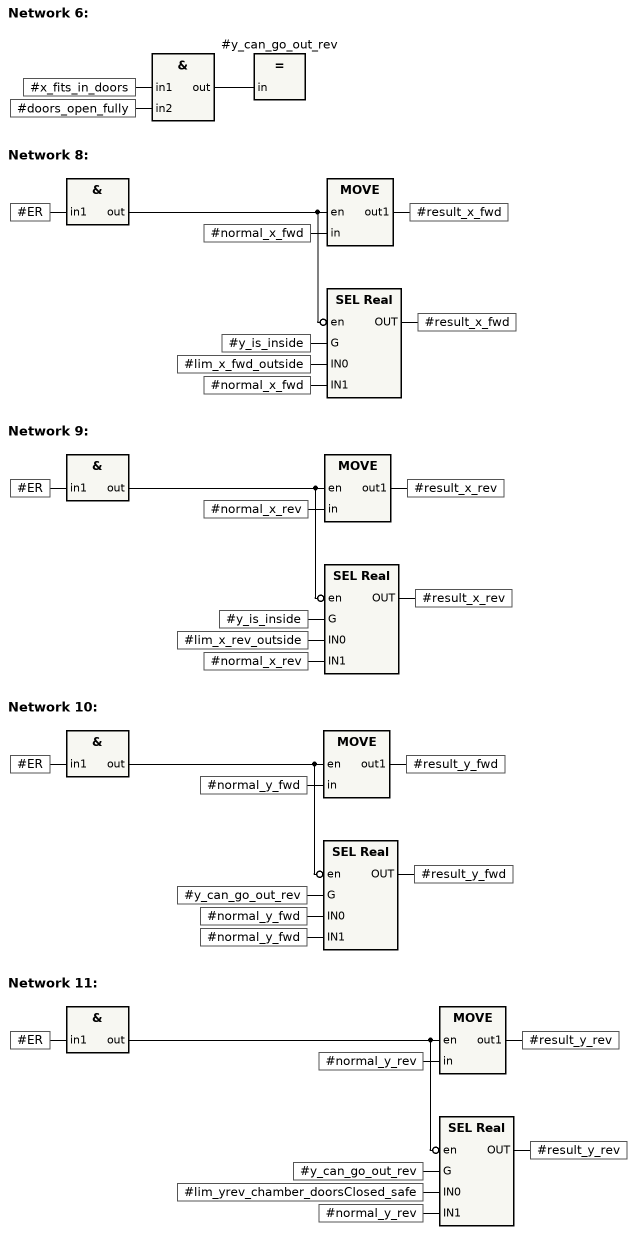
   #y_can_go_out_rev := #x_fits_in_doors AND #doors_open_fully;
END_REGION

REGION Network 8
   IF #ER THEN #result_x_fwd := #normal_x_fwd; END_IF;
   IF NOT #ER THEN
       #result_x_fwd := SEL(G := #y_is_inside, IN0 := #lim_x_fwd_outside, IN1 := #normal_x_fwd);
   END_IF;
END_REGION

REGION Network 9
   IF #ER THEN #result_x_rev := #normal_x_rev; END_IF;
   IF NOT #ER THEN
       #result_x_rev := SEL(G := #y_is_inside, IN0 := #lim_x_rev_outside, IN1 := #normal_x_rev);
   END_IF;
END_REGION

REGION Network 10
   IF #ER THEN #result_y_fwd := #normal_y_fwd; END_IF;
   IF NOT #ER THEN
       #result_y_fwd := SEL(G := #y_can_go_out_rev, IN0 := #normal_y_fwd, IN1 := #normal_y_fwd);
   END_IF;
END_REGION

REGION Network 11
   IF #ER THEN #result_y_rev := #normal_y_rev; END_IF;
   IF NOT #ER THEN
       #result_y_rev := SEL(G := #y_can_go_out_rev, IN0 := #lim_yrev_chamber_doorsClosed_safe, IN1 := #normal_y_rev);
   END_IF;
END_REGION
END_FUNCTION_BLOCK

FUNCTION_BLOCK "_DOOORS_fb"   // FB72, FBD
{ S7_Optimized_Access := 'TRUE' }
VERSION : 0.1
// stored: AutoNumber true, IsIECCheckEnabled false, IsRetainMemResEnabled false, MemoryReserve 100, SetENOAutomatically false, UDAEnableTagReadback false
   VAR_INPUT
      xBtnOpen : Bool;
      xBtnClose : Bool;
      allowedNotAuto : Bool;
      allowedCloseLightBrrier : Bool;
      allowedCloseManipulator : Bool;
      xClosed : Bool;
      xOpen : Bool;
   END_VAR
   VAR_OUTPUT
      yCmdOpen : Bool;
      yCmdClose : Bool;
      sOpen : Bool;
      sClosed : Bool;
      wn_Auto : Bool;
      wnLightbarrier : Bool;
      wnManipulatorClose : Bool;
   END_VAR
   VAR_IN_OUT
      yBeepCosedResetMe : Bool;
   END_VAR
   VAR
      memOpen : Bool;
      memClosed : Bool;
      memopn : Bool;
      memopn1 : Bool;
      memClosed1 : Bool;
   END_VAR
   VAR_TEMP   // added for the SCL form of the ladder/FBD networks
      _w1 : Bool;
      _w2 : Bool;
   END_VAR
BEGIN

REGION Network 1
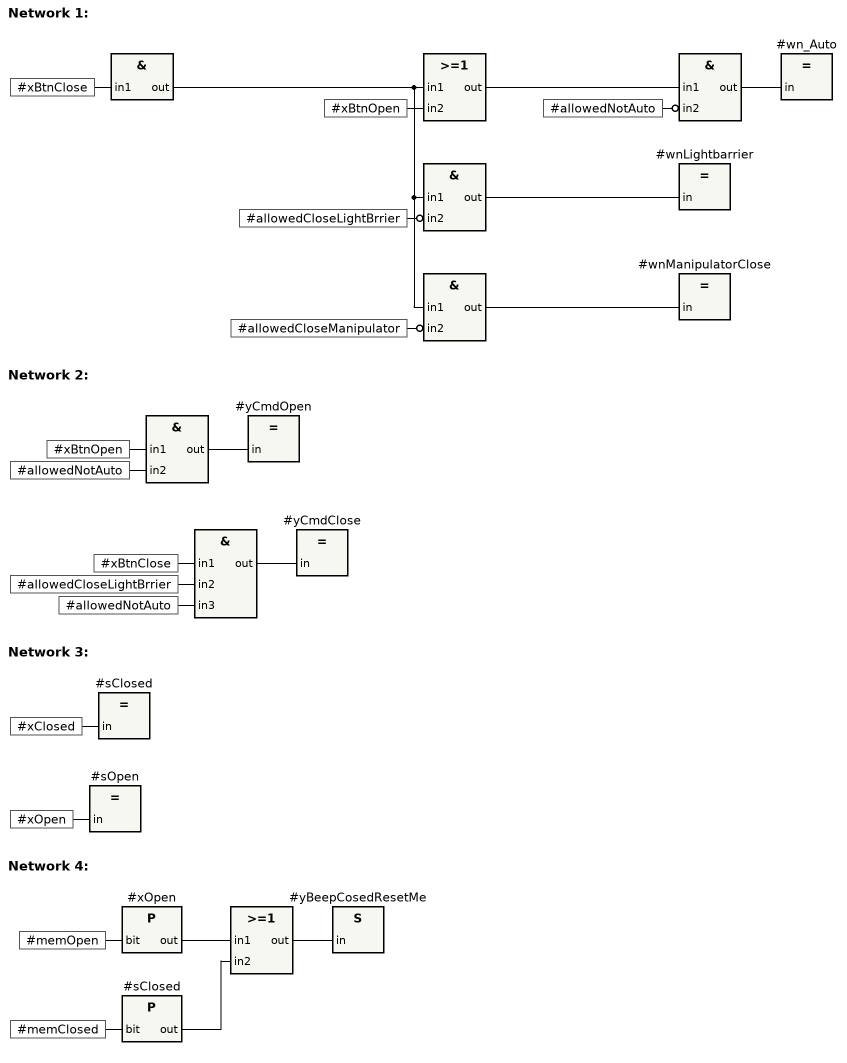
   #wn_Auto := (#xBtnClose OR #xBtnOpen) AND NOT #allowedNotAuto;
   #wnLightbarrier := #xBtnClose AND NOT #allowedCloseLightBrrier;
   #wnManipulatorClose := #xBtnClose AND NOT #allowedCloseManipulator;
END_REGION

REGION Network 2
   #yCmdOpen := #xBtnOpen AND #allowedNotAuto;
   #yCmdClose := #xBtnClose AND #allowedCloseLightBrrier AND #allowedNotAuto;
END_REGION

REGION Network 3
   #sClosed := #xClosed;
   #sOpen := #xOpen;
END_REGION

REGION Network 4
   #_w1 := #xOpen AND NOT #memOpen;   // rising edge of #xOpen
   #memOpen := #xOpen;
   #_w2 := #sClosed AND NOT #memClosed;   // rising edge of #sClosed
   #memClosed := #sClosed;
   IF #_w1 OR #_w2 THEN #yBeepCosedResetMe := TRUE; END_IF;
END_REGION
END_FUNCTION_BLOCK

ORGANIZATION_BLOCK "Cyclic interrupt_comms_50ms"   // OB30, FBD, CyclicInterrupt
{ S7_Optimized_Access := 'TRUE' }
VERSION : 0.1
// stored: AutoNumber true, IsIECCheckEnabled false, SetENOAutomatically false
   VAR_INPUT
      Initial_Call : Bool;
      Event_Count : Int;
   END_VAR
BEGIN

REGION Network 1
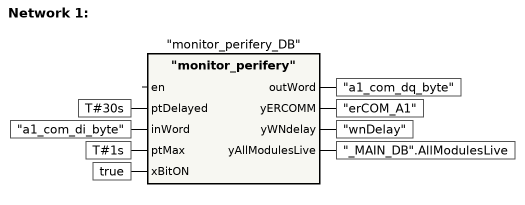
   "monitor_perifery_DB"(ptDelayed := T#30s,   // "monitor_perifery"
                         inWord := "a1_com_di_byte",
                         ptMax := T#1s,
                         xBitON := true,
                         outWord => "a1_com_dq_byte",
                         yERCOMM => "erCOM_A1",
                         yWNdelay => "wnDelay",
                         yAllModulesLive => "_MAIN_DB".AllModulesLive);
END_REGION
END_ORGANIZATION_BLOCK

FUNCTION_BLOCK "monitor_perifery"   // FB55, FBD
{ S7_Optimized_Access := 'TRUE' }
VERSION : 0.1
// stored: AutoNumber true, IsIECCheckEnabled false, IsRetainMemResEnabled false, MemoryReserve 100, SetENOAutomatically false, UDAEnableTagReadback false
   VAR_INPUT
      ptDelayed : Time := T#1m;
      inWord : Byte;
      ptMax : Time := T#300ms;
      xBitON : Bool;
   END_VAR
   VAR_OUTPUT
      outWord : Byte;
      yERCOMM : Bool;
      yWNdelay : Bool;
      yAllModulesLive : Bool;
   END_VAR
   VAR
      IEC_Timer_0_Instance { S7_SetPoint := 'True'} : TON_TIME;
      startup { S7_SetPoint := 'True'} : TON_TIME;
      delayPassed : Bool;
   END_VAR
BEGIN

REGION Network 1
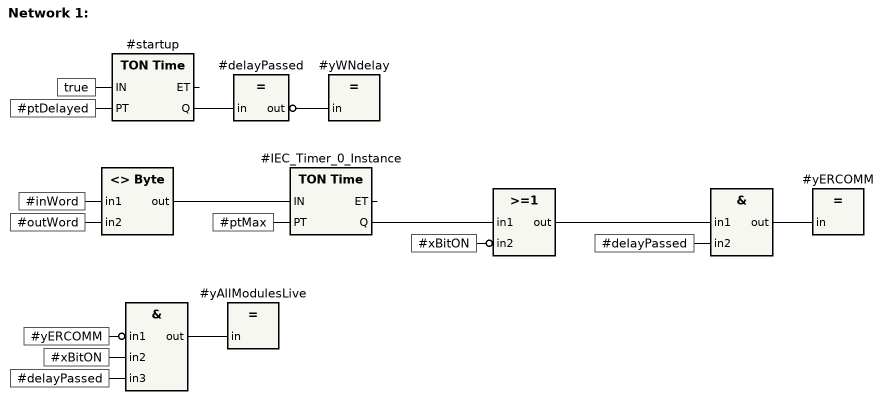
   #startup(IN := true, PT := #ptDelayed);   // TON
   #delayPassed := #startup.Q;
   #yWNdelay := NOT #startup.Q;
   #IEC_Timer_0_Instance(IN := #inWord <> #outWord, PT := #ptMax);   // TON
   #yERCOMM := (#IEC_Timer_0_Instance.Q OR NOT #xBitON) AND #delayPassed;
   #yAllModulesLive := NOT #yERCOMM AND #xBitON AND #delayPassed;
END_REGION

REGION Network 2 (SCL)
   IF (#inWord = #outWord) THEN
       IF #outWord < 100 THEN
           #outWord := #outWord + 1;
       ELSE
           #outWord := 1;
       END_IF;
   END_IF;
END_REGION
END_FUNCTION_BLOCK

FUNCTION_BLOCK "LIVE_BLINK_MONITOR_TESTER"   // FB66, FBD
{ S7_Optimized_Access := 'TRUE' }
VERSION : 0.1
// stored: AutoNumber true, IsIECCheckEnabled false, IsRetainMemResEnabled false, MemoryReserve 100, SetENOAutomatically false, UDAEnableTagReadback false
   VAR_OUTPUT
      flashing : Bool;
      high : Bool;
   END_VAR
   VAR
      BLINKER_Instance { S7_SetPoint := 'True'} : "BLINKER";
      run : Bool;
      blink_t_on : Time;
      blink_t_off : Time;
      run_t_on : Time;
      run_t_off : Time;
      blink_run { S7_SetPoint := 'True'} : "BLINKER";
      test_problems : Bool;
   END_VAR
BEGIN

REGION Network 1
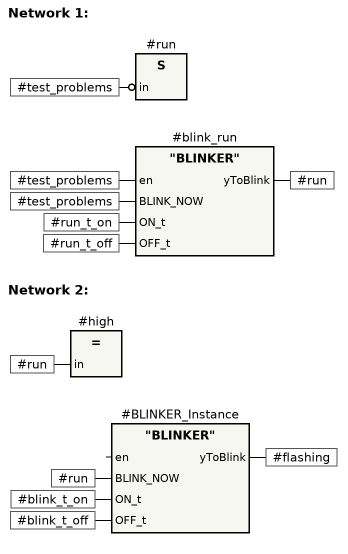
   IF NOT #test_problems THEN #run := TRUE; END_IF;
   IF #test_problems THEN
       #blink_run(BLINK_NOW := #test_problems, ON_t := #run_t_on, OFF_t := #run_t_off, yToBlink => #run);   // "BLINKER"
   END_IF;
END_REGION

REGION Network 2
   #high := #run;
   #BLINKER_Instance(BLINK_NOW := #run, ON_t := #blink_t_on, OFF_t := #blink_t_off, yToBlink => #flashing);   // "BLINKER"
END_REGION
END_FUNCTION_BLOCK

FUNCTION "DINTinSeconds_to_time" : Void   // FC9, FBD
{ S7_Optimized_Access := 'TRUE' }
VERSION : 0.1
// stored: AutoNumber true, IsIECCheckEnabled false, SetENOAutomatically false, UDAEnableTagReadback false
   VAR_INPUT
      in : DInt;
   END_VAR
   VAR_OUTPUT
      out : Time;
   END_VAR
   VAR_TEMP
      pt_dint_by_1000 : DInt;
   END_VAR
BEGIN

REGION Network 1
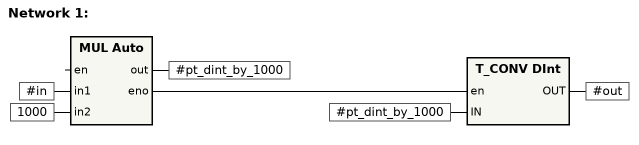
   #pt_dint_by_1000 := #in * 1000;
   T_CONV(IN := #pt_dint_by_1000, OUT => #out);
END_REGION
END_FUNCTION

FUNCTION_BLOCK "SR_CLK"   // FB9, FBD
{ S7_Optimized_Access := 'TRUE' }
VERSION : 0.1
// stored: AutoNumber true, IsIECCheckEnabled false, IsRetainMemResEnabled false, MemoryReserve 100, SetENOAutomatically false, UDAEnableTagReadback false
   VAR_INPUT
      CLK : Bool;
   END_VAR
   VAR_IN_OUT
      Q : Bool;
   END_VAR
   VAR
      mem_R : Bool;
      mem_S : Bool;
   END_VAR
   VAR_TEMP   // added for the SCL form of the ladder/FBD networks
      _w1 : Bool;
      _w2 : Bool;
   END_VAR
BEGIN

REGION Network 1
